Staubli VAL3: ClsPage.pgx

program ClsPage(num x_n1x (dimensions=1), num x_n1y (dimensions=1), num x_n2x (dimensions=1), num x_n2y (dimensions=1))
  local num l_nI
  local num l_nJ
begin
  for l_nI=x_n1x to x_n2x
    for l_nJ=x_n1y to x_n2y
      gotoxy(l_nI,l_nJ)
      put(" ")
    endFor
  endFor
end
